{attribute addProperty BoxType "EPP2339-0003-0016"}
{attribute addProperty Id "DI_Inputs_ChannelAT %I*ARRAY[0..1] OF DI_Inputs_Channel_595007DD176220DO_Outputs_ChannelAT %Q*ARRAY[0..1] OF DO_Outputs_Channel_33B76376128160WcStateAT %I*WcState_F855686C1620InfoDataAT %I*InfoData_BC63D37F80100"}
{attribute addProperty CRC "294202964"}
{attribute addProperty SizeInBites "400"}
{attribute addProperty SizeInBytes "50"}
TYPE EPP2339_CCF4B643 :
STRUCT
	{attribute addProperty Name "DI_Inputs_Channel"}
	DI_Inputs_Channel : ARRAY[0..1] OF DI_Inputs_Channel_595007DD;
	{attribute addProperty Name "DO_Outputs_Channel"}
	DO_Outputs_Channel : ARRAY[0..1] OF DO_Outputs_Channel_33B76376;
	{attribute addProperty Name "WcState"}
	WcState : WcState_F855686C;
	{attribute addProperty Name "InfoData"}
	InfoData : InfoData_BC63D37F;
END_STRUCT
END_TYPE

(* stored: Version 1.2.0.0, ProductVersion 3.1.4024.9
   DUT EPP2339_CCF4B643: Id {6776ceb9-51a7-4aa5-8909-16e568655af8} *)
